DATA_BLOCK "LBP_Axis30"   // DB60
TITLE = Axis-specific signals / Signaux spécifiques à un axe
{ S7_Optimized_Access := 'FALSE' }
AUTHOR : SINUMERIK
FAMILY : SINUMERIK_ONE
VERSION : 6.24
// Interface between user program and axis/spindle, contains signals from/to axis/spindle 30 / Interface entre programme utilisateur et axe/broche, contient des signaux de/vers axe/broche 30
// stored: AutoNumber false, InstanceOfName LBP_typeAxisX, InstanceOfType UDT
"LBP_typeAxisX"
BEGIN
END_DATA_BLOCK

DATA_BLOCK "LBP_Axis31"   // DB61
TITLE = Axis-specific signals / Signaux spécifiques à un axe
{ S7_Optimized_Access := 'FALSE' }
AUTHOR : SINUMERIK
FAMILY : SINUMERIK_ONE
VERSION : 6.24
// Interface between user program and axis/spindle, contains signals from/to axis/spindle 31 / Interface entre programme utilisateur et axe/broche, contient des signaux de/vers axe/broche 31
// stored: AutoNumber false, InstanceOfName LBP_typeAxisX, InstanceOfType UDT
"LBP_typeAxisX"
BEGIN
END_DATA_BLOCK

DATA_BLOCK "LBP_Chan1"   // DB21
TITLE = Channel-specific signals / Signaux spécifiques à un canal
{ S7_Optimized_Access := 'FALSE' }
AUTHOR : SINUMERIK
FAMILY : SINUMERIK_ONE
VERSION : 6.24
// Interface between user program and channel, contains signals from/to channel 1 / Interface entre programme utilisateur et canal, contient des signaux de/vers canal 1
// stored: AutoNumber false, InstanceOfName LBP_typeChanX, InstanceOfType UDT
"LBP_typeChanX"
BEGIN
END_DATA_BLOCK

DATA_BLOCK "LBP_Chan10"   // DB30
TITLE = Channel-specific signals / Signaux spécifiques à un canal
{ S7_Optimized_Access := 'FALSE' }
AUTHOR : SINUMERIK
FAMILY : SINUMERIK_ONE
VERSION : 6.24
// Interface between user program and channel, contains signals from/to channel 10 / Interface entre programme utilisateur et canal, contient des signaux de/vers canal 10
// stored: AutoNumber false, InstanceOfName LBP_typeChanX, InstanceOfType UDT
"LBP_typeChanX"
BEGIN
END_DATA_BLOCK

DATA_BLOCK "LBP_Chan2"   // DB22
TITLE = Channel-specific signals / Signaux spécifiques à un canal
{ S7_Optimized_Access := 'FALSE' }
AUTHOR : SINUMERIK
FAMILY : SINUMERIK_ONE
VERSION : 6.24
// Interface between user program and channel, contains signals from/to channel 2 / Interface entre programme utilisateur et canal, contient des signaux de/vers canal 2
// stored: AutoNumber false, InstanceOfName LBP_typeChanX, InstanceOfType UDT
"LBP_typeChanX"
BEGIN
END_DATA_BLOCK

DATA_BLOCK "LBP_Chan3"   // DB23
TITLE = Channel-specific signals / Signaux spécifiques à un canal
{ S7_Optimized_Access := 'FALSE' }
AUTHOR : SINUMERIK
FAMILY : SINUMERIK_ONE
VERSION : 6.24
// Interface between user program and channel, contains signals from/to channel 3 / Interface entre programme utilisateur et canal, contient des signaux de/vers canal 3
// stored: AutoNumber false, InstanceOfName LBP_typeChanX, InstanceOfType UDT
"LBP_typeChanX"
BEGIN
END_DATA_BLOCK

DATA_BLOCK "LBP_Chan4"   // DB24
TITLE = Channel-specific signals / Signaux spécifiques à un canal
{ S7_Optimized_Access := 'FALSE' }
AUTHOR : SINUMERIK
FAMILY : SINUMERIK_ONE
VERSION : 6.24
// Interface between user program and channel, contains signals from/to channel 4 / Interface entre programme utilisateur et canal, contient des signaux de/vers canal 4
// stored: AutoNumber false, InstanceOfName LBP_typeChanX, InstanceOfType UDT
"LBP_typeChanX"
BEGIN
END_DATA_BLOCK

DATA_BLOCK "LBP_Chan5"   // DB25
TITLE = Channel-specific signals / Signaux spécifiques à un canal
{ S7_Optimized_Access := 'FALSE' }
AUTHOR : SINUMERIK
FAMILY : SINUMERIK_ONE
VERSION : 6.24
// Interface between user program and channel, contains signals from/to channel 5 / Interface entre programme utilisateur et canal, contient des signaux de/vers canal 5
// stored: AutoNumber false, InstanceOfName LBP_typeChanX, InstanceOfType UDT
"LBP_typeChanX"
BEGIN
END_DATA_BLOCK

DATA_BLOCK "LBP_Chan6"   // DB26
TITLE = Channel-specific signals / Signaux spécifiques à un canal
{ S7_Optimized_Access := 'FALSE' }
AUTHOR : SINUMERIK
FAMILY : SINUMERIK_ONE
VERSION : 6.24
// Interface between user program and channel, contains signals from/to channel 6 / Interface entre programme utilisateur et canal, contient des signaux de/vers canal 6
// stored: AutoNumber false, InstanceOfName LBP_typeChanX, InstanceOfType UDT
"LBP_typeChanX"
BEGIN
END_DATA_BLOCK

DATA_BLOCK "LBP_Chan7"   // DB27
TITLE = Channel-specific signals / Signaux spécifiques à un canal
{ S7_Optimized_Access := 'FALSE' }
AUTHOR : SINUMERIK
FAMILY : SINUMERIK_ONE
VERSION : 6.24
// Interface between user program and channel, contains signals from/to channel 7 / Interface entre programme utilisateur et canal, contient des signaux de/vers canal 7
// stored: AutoNumber false, InstanceOfName LBP_typeChanX, InstanceOfType UDT
"LBP_typeChanX"
BEGIN
END_DATA_BLOCK

DATA_BLOCK "LBP_Chan8"   // DB28
TITLE = Channel-specific signals / Signaux spécifiques à un canal
{ S7_Optimized_Access := 'FALSE' }
AUTHOR : SINUMERIK
FAMILY : SINUMERIK_ONE
VERSION : 6.24
// Interface between user program and channel, contains signals from/to channel 8 / Interface entre programme utilisateur et canal, contient des signaux de/vers canal 8
// stored: AutoNumber false, InstanceOfName LBP_typeChanX, InstanceOfType UDT
"LBP_typeChanX"
BEGIN
END_DATA_BLOCK

DATA_BLOCK "LBP_Chan9"   // DB29
TITLE = Channel-specific signals / Signaux spécifiques à un canal
{ S7_Optimized_Access := 'FALSE' }
AUTHOR : SINUMERIK
FAMILY : SINUMERIK_ONE
VERSION : 6.24
// Interface between user program and channel, contains signals from/to channel 9 / Interface entre programme utilisateur et canal, contient des signaux de/vers canal 9
// stored: AutoNumber false, InstanceOfName LBP_typeChanX, InstanceOfType UDT
"LBP_typeChanX"
BEGIN
END_DATA_BLOCK

DATA_BLOCK "LBP_ConfigData"   // DB7
TITLE = Configuration parameter
{ S7_Optimized_Access := 'FALSE' }
AUTHOR : SINUMERIK
FAMILY : SINUMERIK_ONE
VERSION : 6.14
// Contains parameters for the configuration and initialization of the basic program
// stored: AutoNumber false, InstanceOfName LBP_typeConfigData, InstanceOfType UDT
"LBP_typeConfigData"
BEGIN
END_DATA_BLOCK

DATA_BLOCK "LBP_HMI"   // DB19
TITLE = Operator panel signals / Signaux pupitre opérateur
{ S7_Optimized_Access := 'FALSE' }
AUTHOR : SINUMERIK
FAMILY : SINUMERIK_ONE
VERSION : 6.24
// Interface between user program and operator panel, contains signals from/to the operating software. / Interface entre programme utilisateur et pupitre opérateur, contient des signaux de/vers le logiciel d'exploitation.
// stored: AutoNumber false, InstanceOfName LBP_typeHMI, InstanceOfType UDT
"LBP_typeHMI"
BEGIN
END_DATA_BLOCK

DATA_BLOCK "LBP_ModeGroup"   // DB11
TITLE = Mode group signals / Signaux groupe de modes de fonctionnement
{ S7_Optimized_Access := 'FALSE' }
AUTHOR : SINUMERIK
FAMILY : SINUMERIK_ONE
VERSION : 6.24
// Interface between user program and mode groups, contains signals from/to the NC and operating software / Interface entre programme utilisateur et les groupes de modes de fonctionnement, contient des signaux de/vers le logiciel d'exploitation
// stored: AutoNumber false, InstanceOfName LBP_typeModeGroup, InstanceOfType UDT
"LBP_typeModeGroup"
BEGIN
END_DATA_BLOCK

DATA_BLOCK "LBP_NC"   // DB10
TITLE = NC signals / Signaux CN
{ S7_Optimized_Access := 'FALSE' }
AUTHOR : SINUMERIK
FAMILY : SINUMERIK_ONE
VERSION : 6.24
// Interface between user program and NC, contains signals from/to the NC, PLC and operating software. / Interface entre programme utilisateur et CN, contient des signaux de/vers CN, AP et logiciel d'exploitation.
// stored: AutoNumber false, InstanceOfName LBP_typeNC, InstanceOfType UDT
"LBP_typeNC"
BEGIN
END_DATA_BLOCK

DATA_BLOCK "LBP_OpUnitComm_DB"   // DB70
// stored: InstanceOfName LBP_OpUnitComm, InstanceOfType FB
"LBP_OpUnitComm"
   // VAR_OUTPUT
   //    Error : Bool;
   //    Status : Word;
   // END_VAR
   // VAR_IN_OUT
   //    Config : Variant;
   // END_VAR
   // VAR
   //    s_OpUnitConnInstance { S7_SetPoint := 'True'} : Array[1..6] of "LBP_InternalProc2";
   //    s_OpUnitNumber : UInt;
   //    s_OpUnitHardwareInterfaceId : HW_ANY;
   //    s_OpUnitEnabled : Array[1..6] of Bool;
   //    s_OpUnitConfig { S7_SetPoint := 'True'} : Array[1..6] of "LBP_typeInternal1";
   //    s_OpUnitControlMcp : Array[1..5] of Struct
   //       active : Bool;
   //       stop : Bool;
   //       notSend : Bool;
   //       connected : Bool;
   //       warning : Bool;
   //       error : Bool;
   //       status : Word;
   //       info : Word;
   //       alert : Bool;
   //       alertDelay { S7_SetPoint := 'True'} : TON_TIME;
   //    END_STRUCT;
   //    s_OpUnitControlIdent : Struct
   //       strobe : Bool;
   //       busAddress : USInt;
   //       modeDck : Bool;
   //       numberOfInputBytes : UInt;
   //       numberOfOutputBytes : UInt;
   //       mcpType : Word;
   //       done : Bool;
   //       error : Bool;
   //       status : Word;
   //       info : Word;
   //    END_STRUCT;
   //    s_OpUnitData : Array[1..6] of Struct
   //       connect : Bool;
   //       ident : Bool;
   //       notSend : Bool;
   //       busy : Bool;
   //       connected : Bool;
   //       warning : Bool;
   //       error : Bool;
   //       identReady : Bool;
   //       reconnect : Bool;
   //       status : Word;
   //       errorInfo : Word;
   //       mcpType : Word;
   //       mcpDipFixes : Word;
   //       numberOfOutputBytes : UInt;
   //       numberOfInputBytes : UInt;
   //       numberOfHandwheels : UInt;
   //       handwheelRecent : Bool;
   //       handwheelPulses1 : Int;
   //       handwheelPulses2 : Int;
   //       handwheelStopped1 : Bool;
   //       handwheelStopped2 : Bool;
   //       reconnectTimer { S7_SetPoint := 'True'} : TON_TIME;
   //       reconnectCounter : UInt;
   //    END_STRUCT;
   //    s_init : Bool;
   //    statReadWriteRecordActive : Bool;
   //    statReadWriteRecordComplete : Bool;
   //    statReadWriteRecordAbort : Bool;
   //    statReadWriteRecordMcp : UInt;
   //    statReadWriteRecordTimeout : TON_TIME;
   //    statReadWriteRecordData { S7_SetPoint := 'True'} : "LBP_typeInternal5";
   // END_VAR
BEGIN
END_DATA_BLOCK

DATA_BLOCK "LBP_TMLoad"   // DB71
TITLE = Tool management / Gestion des outils
{ S7_Optimized_Access := 'FALSE' }
AUTHOR : SINUMERIK
FAMILY : SINUMERIK_ONE
VERSION : 6.24
// Interface between user program and tool management, contains signals from/to Load/Unload magazine / Interface entre programme utilisateur et gestion d'outil, contient des signaux de/vers Chargement/déchargement de magasin
// stored: AutoNumber false, InstanceOfName LBP_typeTMLoad, InstanceOfType UDT
"LBP_typeTMLoad"
BEGIN
END_DATA_BLOCK

DATA_BLOCK "LBP_TMLoadMT"   // DB1071
TITLE = Tool management / Gestion des outils
{ S7_Optimized_Access := 'FALSE' }
AUTHOR : SINUMERIK
FAMILY : SINUMERIK_ONE
VERSION : 6.24
// Interface between user program and tool management, contains signals from/to Load/Unload magazine (multitool). / Interface entre programme utilisateur et gestion d'outil, contient des signaux de/vers Chargement/déchargement de magasin (Multitool).
// stored: AutoNumber false, InstanceOfName LBP_typeTMLoadMT, InstanceOfType UDT
"LBP_typeTMLoadMT"
BEGIN
END_DATA_BLOCK

DATA_BLOCK "LBP_TMSpindle"   // DB72
TITLE = Tool management / Gestion des outils
{ S7_Optimized_Access := 'FALSE' }
AUTHOR : SINUMERIK
FAMILY : SINUMERIK_ONE
VERSION : 6.24
// Interface between user program and tool management, contains signals for spindle as change position. / Interface entre programme utilisateur et gestion d'outil, contient des signaux pour broche en tant que position de changement.
// stored: AutoNumber false, InstanceOfName LBP_typeTMSpindle, InstanceOfType UDT
"LBP_typeTMSpindle"
BEGIN
END_DATA_BLOCK

DATA_BLOCK "LBP_TMSpindleMT"   // DB1072
TITLE = Tool management / Gestion des outils
{ S7_Optimized_Access := 'FALSE' }
AUTHOR : SINUMERIK
FAMILY : SINUMERIK_ONE
VERSION : 6.24
// Interface between user program and tool management, contains signals for spindle as change position (multitool). / Interface entre programme utilisateur et gestion d'outil, contient des signaux pour broche en tant que position de changement (Multitool).
// stored: AutoNumber false, InstanceOfName LBP_typeTMSpindleMT, InstanceOfType UDT
"LBP_typeTMSpindleMT"
BEGIN
END_DATA_BLOCK

DATA_BLOCK "LBP_TMTurret"   // DB73
TITLE = Tool management / Gestion des outils
{ S7_Optimized_Access := 'FALSE' }
AUTHOR : SINUMERIK
FAMILY : SINUMERIK_ONE
VERSION : 6.24
// Interface between user program and tool management, contains signals for turret. / Interface entre programme utilisateur et gestion d'outil, contient des signaux pour tourelle.
// stored: AutoNumber false, InstanceOfName LBP_typeTMTurret, InstanceOfType UDT
"LBP_typeTMTurret"
BEGIN
END_DATA_BLOCK

DATA_BLOCK "LBP_TMTurretMT"   // DB1073
TITLE = Tool management / Gestion des outils
{ S7_Optimized_Access := 'FALSE' }
AUTHOR : SINUMERIK
FAMILY : SINUMERIK_ONE
VERSION : 6.24
// Interface between user program and tool management, contains signals for turret (multitool). / Interface entre programme utilisateur et gestion d'outil, contient des signaux pour tourelle (Multitool).
// stored: AutoNumber false, InstanceOfName LBP_typeTMTurretMT, InstanceOfType UDT
"LBP_typeTMTurretMT"
BEGIN
END_DATA_BLOCK

DATA_BLOCK "LBP_Internal2"   // DB25001
TITLE = Internal DB for basic program / DB interne pour programme de base
// DB only for internal use in the basic program / DB réservé à l'utilisation interne dans le programme de base
// stored: InstanceOfName LBP_InternalProc7, InstanceOfType FB
"LBP_InternalProc7"
   // VAR_OUTPUT
   //    error { ExternalAccessible := 'False'; ExternalVisible := 'False'; ExternalWritable := 'False'} : Bool;
   // END_VAR
   // VAR
   //    statTimer1 { ExternalAccessible := 'False'; ExternalVisible := 'False'; ExternalWritable := 'False'} : Array[1..8] of IEC_TIMER;
   //    statTimer2 { ExternalAccessible := 'False'; ExternalVisible := 'False'; ExternalWritable := 'False'} : Array[1..8] of IEC_TIMER;
   //    statTimerActivationImmediately { ExternalAccessible := 'False'; ExternalVisible := 'False'; ExternalWritable := 'False'} : Array[1..8] of IEC_TIMER;   // Delay time for immediate activation / Temporisation pour activation immédiate
   //    statActivationImmediately { ExternalAccessible := 'False'; ExternalVisible := 'False'; ExternalWritable := 'False'} : Array[1..8] of Bool;
   //    statImpReloadT2 { ExternalAccessible := 'False'; ExternalVisible := 'False'; ExternalWritable := 'False'} : Array[1..8] of R_TRIG;
   //    statMcp1 { ExternalAccessible := 'False'; ExternalVisible := 'False'; ExternalWritable := 'False'} : Array[0..1, 0..7] of Byte;   // Image of mcp1 to detect any changes / Image de la mcp1 pour comparaison
   //    statMcp2 { ExternalAccessible := 'False'; ExternalVisible := 'False'; ExternalWritable := 'False'} : Array[0..1, 0..7] of Byte;   // Image of mcp2 to detect any changes / Image de la mcp2 pour comparaison
   //    statTimerDataTranfer { ExternalAccessible := 'False'; ExternalVisible := 'False'; ExternalWritable := 'False'} : IEC_TIMER;
   //    statChanInReset { ExternalAccessible := 'False'; ExternalVisible := 'False'; ExternalWritable := 'False'} : Array[1..10] of Bool;
   //    statAktProfile { ExternalAccessible := 'False'; ExternalVisible := 'False'; ExternalWritable := 'False'} : Struct
   //       ESaveOn : Bool;   // Activate energy-saving profile immediately / Activer immédiatement le profil d'économie d'énergie
   //       ReloadT2 : Bool;   // Reload Prewarning time (T2) / Recharger temps de préavis (T2)
   //       res0_2 : Bool;
   //       res0_3 : Bool;
   //       res0_4 : Bool;
   //       res0_5 : Bool;
   //       res0_6 : Bool;
   //       res0_7 : Bool;
   //       HmiESaveOn : Bool;   // HMI->PLC: Activate energy-saving profile immediately / IHM->AP : activer immédiatement le profil d'économie d'énergie
   //       res1_1 : Bool;
   //       res1_2 : Bool;
   //       res1_3 : Bool;
   //       res1_4 : Bool;
   //       res1_5 : Bool;
   //       res1_6 : Bool;
   //       res1_7 : Bool;
   //       MasterCompSig : Bool;   // Master computer signal / Signal ordinateur maître
   //       PlcUserSig : Bool;   // PLC user signal / AP signal utilisateur
   //       res2_2 : Bool;
   //       res2_3 : Bool;
   //       res2_4 : Bool;
   //       res2_5 : Bool;
   //       res2_6 : Bool;
   //       res2_7 : Bool;
   //       res3 : Byte;
   //       ESaveIsOn : Bool;   // Energy-saving state active / État économie d'énergie actif
   //       T1Expired : Bool;   // Activation time T1 expired / Temps d'activation T1 écoulé
   //       res4_2 : Bool;
   //       res4_3 : Bool;
   //       res4_4 : Bool;
   //       res4_5 : Bool;
   //       res4_6 : Bool;
   //       res4_7 : Bool;
   //       res5 : Byte;
   //       ActValT1 : Int;   // T1 current value / T1 valeur réelle
   //       ActValT2 : Int;   // T2 current value / T2 valeur réelle
   //       ESaveValid : Bool;   // HMI->PLC: Energy-saving profile valid / IHM->AP : profil d'économie d'énergie valide
   //       ESaveOff : Bool;   // HMI->PLC: Deactivate energy-saving profileblock energy-saving profile / IHM->AP : désactiver/bloquer le profil d'économie d'énergie
   //       res10_2 : Bool;
   //       res10_3 : Bool;
   //       res10_4 : Bool;
   //       res10_5 : Bool;
   //       res10_6 : Bool;
   //       res10_7 : Bool;
   //       CondOpPanel : Bool;   // HMI->PLC: Operator panel / IHM->AP : pupitre opérateur
   //       CondDataTransfer : Bool;   // HMI->PLC: Data transfer / IHM->AP : transmission de données
   //       CondWindowChange : Bool;   // HMI->PLC: Window change / IHM->AP : changement de fenêtre
   //       res11_3 : Bool;
   //       res11_4 : Bool;
   //       res11_5 : Bool;
   //       res11_6 : Bool;
   //       res11_7 : Bool;
   //       CondMCP : Bool;   // HMI->PLC: Machine control panel / IHM->AP : pupitre opérateur machine
   //       res12_1 : Bool;
   //       res12_2 : Bool;
   //       res12_3 : Bool;
   //       res12_4 : Bool;
   //       res12_5 : Bool;
   //       res12_6 : Bool;
   //       res12_7 : Bool;
   //       CondNcChan1 : Bool;   // HMI->PLC: NC channel 1 in reset / IHM->AP : canal CN 1 en Reset
   //       CondNcChan2 : Bool;   // HMI->PLC: NC channel 2 in reset / IHM->AP : canal CN 2 en Reset
   //       CondNcChan3 : Bool;   // HMI->PLC: NC channel 3 in reset / IHM->AP : canal CN 3 en Reset
   //       CondNcChan4 : Bool;   // HMI->PLC: NC channel 4 in reset / IHM->AP : canal CN 4 en Reset
   //       CondNcChan5 : Bool;   // HMI->PLC: NC channel 5 in reset / IHM->AP : canal CN 5 en Reset
   //       CondNcChan6 : Bool;   // HMI->PLC: NC channel 6 in reset / IHM->AP : canal CN 6 en Reset
   //       CondNcChan7 : Bool;   // HMI->PLC: NC channel 7 in reset / IHM->AP : canal CN 7 en Reset
   //       CondNcChan8 : Bool;   // HMI->PLC: NC channel 8 in reset / IHM->AP : canal CN 8 en Reset
   //       CondNcChan9 : Bool;   // HMI->PLC: NC channel 9 in reset / IHM->AP : canal CN 9 en Reset
   //       CondNcChan10 : Bool;   // HMI->PLC: NC channel 10 in reset / IHM->AP : canal CN 10 en Reset
   //       res14_2 : Bool;
   //       res14_3 : Bool;
   //       res14_4 : Bool;
   //       res14_5 : Bool;
   //       res14_6 : Bool;
   //       res14_7 : Bool;
   //       CondMasterCompSig : Bool;   // HMI->PLC: Master computer signal / IHM->AP : signal ordinateur maître
   //       CondPlcUserSig : Bool;   // HMI->PLC: PLC user signal / IHM->AP : signal utilisateur AP
   //       res15_2 : Bool;
   //       res15_3 : Bool;
   //       res15_4 : Bool;
   //       res15_5 : Bool;
   //       res15_6 : Bool;
   //       res15_7 : Bool;
   //       PresetT1 : Int;   // HMI->PLC: Activation time T1 / IHM->AP : temps d'activation T1
   //       PresetT2 : Int;   // HMI->PLC: Activation time T2 / IHM->AP : temps d'activation T2
   //    END_STRUCT;
   // END_VAR
BEGIN
END_DATA_BLOCK

DATA_BLOCK "LBP_Internal3"   // DB25002
TITLE = Internal DB for basic program / DB interne pour programme de base
// DB only for internal use in the basic program / DB réservé à l'utilisation interne dans le programme de base
// stored: InstanceOfName LBP_InternalProc8, InstanceOfType FB
"LBP_InternalProc8"
   // VAR
   //    statPlcCtrlsNm1 { ExternalAccessible := 'False'; ExternalVisible := 'False'; ExternalWritable := 'False'} : Bool;
   //    statDateAndTime { ExternalAccessible := 'False'; ExternalVisible := 'False'; ExternalWritable := 'False'} : Date_And_Time;
   //    statLastSecond { ExternalAccessible := 'False'; ExternalVisible := 'False'; ExternalWritable := 'False'} : Byte;
   // END_VAR
BEGIN
END_DATA_BLOCK

DATA_BLOCK "LBP_Internal9"   // DB25005
TITLE = Internal DB for basic program / DB interne pour programme de base
// DB only for internal use in the basic program / DB réservé à l'utilisation interne dans le programme de base
// stored: InstanceOfName LBP_InternalProc9, InstanceOfType FB
"LBP_InternalProc9"
   // VAR
   //    statSymbols { ExternalAccessible := 'False'; ExternalVisible := 'False'; ExternalWritable := 'False'} : Array[0..31] of WString;
   //    statResolvedSymbols { ExternalAccessible := 'False'; ExternalVisible := 'False'; ExternalWritable := 'False'} : Array[0..31] of ResolvedSymbol;
   //    InstResolveSymbols { ExternalAccessible := 'False'; ExternalVisible := 'False'; ExternalWritable := 'False'} : ResolveSymbols;
   //    statDestOffsets { ExternalAccessible := 'False'; ExternalVisible := 'False'; ExternalWritable := 'False'} : Array[0..31] of DInt;
   //    statResolveExecute { ExternalAccessible := 'False'; ExternalVisible := 'False'; ExternalWritable := 'False'} : Bool;
   //    statResolveProcessing { ExternalAccessible := 'False'; ExternalVisible := 'False'; ExternalWritable := 'False'} : Bool;
   //    statResolveError { ExternalAccessible := 'False'; ExternalVisible := 'False'; ExternalWritable := 'False'} : Bool;
   //    statResolveStatus { ExternalAccessible := 'False'; ExternalVisible := 'False'; ExternalWritable := 'False'} : Word;
   //    statReResolveNeeded { ExternalAccessible := 'False'; ExternalVisible := 'False'; ExternalWritable := 'False'} : Array[0..31] of Bool;
   // END_VAR
BEGIN
END_DATA_BLOCK

DATA_BLOCK "LBP_InternalDB1020"   // DB1020
TITLE = Internal DB for basic program / DB interne pour programme de base
// DB only for internal use in the basic program / DB réservé à l'utilisation interne dans le programme de base
// stored: AutoNumber false, InstanceOfName LBP_InternalFB1020, InstanceOfType FB
"LBP_InternalFB1020"
   // VAR_INPUT
   //    IN1 : UDInt;
   //    IN2 : UDInt;
   //    IN3 : Word;
   //    IN4 : Variant;
   //    IN5 : Variant;
   //    IN6 : Variant;
   //    IN7 : Variant;
   //    IN8 : Variant;
   //    IN9 : Variant;
   //    IN10 : Variant;
   //    IN11 : Variant;
   //    IN12 : Variant;
   // END_VAR
   // VAR_OUTPUT
   //    OUT1 : Bool;
   //    OUT2 : DWord;
   //    OUT3 : UInt;
   // END_VAR
   // VAR
   //    LBP_AlarmType_ErrMsg { S7_SetPoint := 'True'} : Diag_Alarm;
   //    LBP_AlarmType_OpMsg { S7_SetPoint := 'True'} : Diag_Alarm;
   //    LBP_AlarmType_InfoMsg { S7_SetPoint := 'True'} : Diag_Alarm;
   //    LBP_DB2AlarmType_ErrMsg { S7_SetPoint := 'True'} : Diag_Alarm;
   //    LBP_DB2AlarmType_OpMsg { S7_SetPoint := 'True'} : Diag_Alarm;
   //    LBP_DB2AlarmType_InfoMsg { S7_SetPoint := 'True'} : Diag_Alarm;
   //    LBP_UserAlarmType_ErrMsg { S7_SetPoint := 'True'} : Diag_Alarm;
   //    LBP_UserAlarmType_OpMsg { S7_SetPoint := 'True'} : Diag_Alarm;
   //    LBP_UserAlarmType_InfoMsg { S7_SetPoint := 'True'} : Diag_Alarm;
   //    LBP_UserAlarmType_AckMsg { S7_SetPoint := 'True'} : Diag_Alarm;
   //    s_strct_DB2AddressLastCycle : Struct
   //       LwByteAddress : DInt;
   //       LwBitAddress : DInt;
   //    END_STRUCT;
   //    s_DB2_MaxScanByteUser : DInt;
   //    s_DB7_Params : Struct
   //       MaxAxis : Int;
   //       MaxChan : Int;
   //       MsgUser : Int;
   //       ExtendChanAxMsg : Bool;
   //       ActivChan : Array[1..10] of Bool;
   //       ActivAxis : Array[1..31] of Bool;
   //    END_STRUCT;
   //    s_firstScanFinished : Bool;
   //    s_FC10_Quit : Struct
   //       QuitEdge : Bool;
   //       LwByteAddress : DInt;
   //       DB2ScanFinished : Bool;
   //    END_STRUCT;
   //    s_CounterActiveDB2Alarms : UInt;
   //    s_FC10_ToUserIf_OLD : Bool;
   // END_VAR
BEGIN
END_DATA_BLOCK

DATA_BLOCK "LBP_InternalDB3"   // DB3
TITLE = PLC-Error / Messages / Erreur AP / messages
{ S7_Optimized_Access := 'FALSE' }
AUTHOR : SINUMERIK
FAMILY : SINUMERIK_ONE
VERSION : 6.24
// DB only for internal use in the basic program / DB réservé à l'utilisation interne dans le programme de base
// stored: AutoNumber false, InstanceOfName LBP_typeAlarmMsgs, InstanceOfType UDT
"LBP_typeAlarmMsgs"
BEGIN
END_DATA_BLOCK

DATA_BLOCK "DB_AnalogInputs"   // DB2200
// stored: AutoNumber false, InstanceOfName FB_AnalogInputs, InstanceOfType FB
"FB_AnalogInputs"
BEGIN
END_DATA_BLOCK

DATA_BLOCK "DB_DigitalInputs"   // DB2210
// stored: AutoNumber false, InstanceOfName FB_DigitalInputs, InstanceOfType FB
"FB_DigitalInputs"
BEGIN
END_DATA_BLOCK

DATA_BLOCK "DB_DigitalInputsBW_Station"   // DB2214
// stored: AutoNumber false, InstanceOfName FB_DigitalInputsBW_Station, InstanceOfType FB
"FB_DigitalInputsBW_Station"
BEGIN
END_DATA_BLOCK

DATA_BLOCK "DB_DigitalInputsSonplas"   // DB2211
// stored: AutoNumber false, InstanceOfName FB_DigitalInputsSonplas, InstanceOfType FB
"FB_DigitalInputsSonplas"
BEGIN
END_DATA_BLOCK

DATA_BLOCK "DB_AnalogOutputs"   // DB2113
// stored: AutoNumber false, InstanceOfName FB_AnalogOutputs, InstanceOfType FB
"FB_AnalogOutputs"
BEGIN
END_DATA_BLOCK

DATA_BLOCK "DB_DigitalOutputs"   // DB2103
// stored: AutoNumber false, InstanceOfName FB_DigitalOutputs, InstanceOfType FB
"FB_DigitalOutputs"
BEGIN
END_DATA_BLOCK

DATA_BLOCK "DB_DigitalOutputsSonplas"   // DB2104
// stored: AutoNumber false, InstanceOfName FB_DigitalOutputsSonplas, InstanceOfType FB
"FB_DigitalOutputsSonplas"
BEGIN
END_DATA_BLOCK

DATA_BLOCK "F-DB_DigitalInputs"   // DB110, F_DB
// stored: AutoNumber false, InstanceOfName F-FB_DigitalInput, InstanceOfType FB
"F-FB_DigitalInput"
BEGIN
END_DATA_BLOCK

DATA_BLOCK "F-DB_DigitalOutput"   // DB111, F_DB
// stored: AutoNumber false, InstanceOfName F-FB_DigitalOutput, InstanceOfType FB
"F-FB_DigitalOutput"
BEGIN
END_DATA_BLOCK

DATA_BLOCK "LBP_ReadVar_DB_Axis01_X"   // DB4101
// stored: AutoNumber false, InstanceOfName LBP_ReadVar, InstanceOfType FB
"LBP_ReadVar"
   // VAR_INPUT
   //    Req : Bool;
   //    NumVar : Int;
   //    Addr1 : Variant;
   //    Unit1 : Byte;
   //    Column1 : Word;
   //    Line1 : Word;
   //    Addr2 : Variant;
   //    Unit2 : Byte;
   //    Column2 : Word;
   //    Line2 : Word;
   //    Addr3 : Variant;
   //    Unit3 : Byte;
   //    Column3 : Word;
   //    Line3 : Word;
   //    Addr4 : Variant;
   //    Unit4 : Byte;
   //    Column4 : Word;
   //    Line4 : Word;
   //    Addr5 : Variant;
   //    Unit5 : Byte;
   //    Column5 : Word;
   //    Line5 : Word;
   //    Addr6 : Variant;
   //    Unit6 : Byte;
   //    Column6 : Word;
   //    Line6 : Word;
   //    Addr7 : Variant;
   //    Unit7 : Byte;
   //    Column7 : Word;
   //    Line7 : Word;
   //    Addr8 : Variant;
   //    Unit8 : Byte;
   //    Column8 : Word;
   //    Line8 : Word;
   // END_VAR
   // VAR_OUTPUT
   //    Error : Bool;
   //    NDR : Bool;
   //    State : Word;
   // END_VAR
   // VAR_IN_OUT
   //    RD1 : Variant;
   //    RD2 : Variant;
   //    RD3 : Variant;
   //    RD4 : Variant;
   //    RD5 : Variant;
   //    RD6 : Variant;
   //    RD7 : Variant;
   //    RD8 : Variant;
   // END_VAR
   // VAR
   //    ident : Byte;
   //    regist : Bool;
   //    flanke : Bool;
   //    progtest : Bool;
   //    err_cls_cod : Word;
   //    err_stat : Word;
   //    s_fifoRef : UInt;
   //    s_Reserved1 : Word;
   //    s_Reserved2 : DWord;
   //    s_Reserved3 : DWord;
   // END_VAR
BEGIN
END_DATA_BLOCK

DATA_BLOCK "LBP_ReadVar_DB_Axis02_Y"   // DB4102
// stored: AutoNumber false, InstanceOfName LBP_ReadVar, InstanceOfType FB
"LBP_ReadVar"
   // VAR_INPUT
   //    Req : Bool;
   //    NumVar : Int;
   //    Addr1 : Variant;
   //    Unit1 : Byte;
   //    Column1 : Word;
   //    Line1 : Word;
   //    Addr2 : Variant;
   //    Unit2 : Byte;
   //    Column2 : Word;
   //    Line2 : Word;
   //    Addr3 : Variant;
   //    Unit3 : Byte;
   //    Column3 : Word;
   //    Line3 : Word;
   //    Addr4 : Variant;
   //    Unit4 : Byte;
   //    Column4 : Word;
   //    Line4 : Word;
   //    Addr5 : Variant;
   //    Unit5 : Byte;
   //    Column5 : Word;
   //    Line5 : Word;
   //    Addr6 : Variant;
   //    Unit6 : Byte;
   //    Column6 : Word;
   //    Line6 : Word;
   //    Addr7 : Variant;
   //    Unit7 : Byte;
   //    Column7 : Word;
   //    Line7 : Word;
   //    Addr8 : Variant;
   //    Unit8 : Byte;
   //    Column8 : Word;
   //    Line8 : Word;
   // END_VAR
   // VAR_OUTPUT
   //    Error : Bool;
   //    NDR : Bool;
   //    State : Word;
   // END_VAR
   // VAR_IN_OUT
   //    RD1 : Variant;
   //    RD2 : Variant;
   //    RD3 : Variant;
   //    RD4 : Variant;
   //    RD5 : Variant;
   //    RD6 : Variant;
   //    RD7 : Variant;
   //    RD8 : Variant;
   // END_VAR
   // VAR
   //    ident : Byte;
   //    regist : Bool;
   //    flanke : Bool;
   //    progtest : Bool;
   //    err_cls_cod : Word;
   //    err_stat : Word;
   //    s_fifoRef : UInt;
   //    s_Reserved1 : Word;
   //    s_Reserved2 : DWord;
   //    s_Reserved3 : DWord;
   // END_VAR
BEGIN
END_DATA_BLOCK

DATA_BLOCK "LBP_ReadVar_DB_Axis03_ZM"   // DB4103
// stored: AutoNumber false, InstanceOfName LBP_ReadVar, InstanceOfType FB
"LBP_ReadVar"
   // VAR_INPUT
   //    Req : Bool;
   //    NumVar : Int;
   //    Addr1 : Variant;
   //    Unit1 : Byte;
   //    Column1 : Word;
   //    Line1 : Word;
   //    Addr2 : Variant;
   //    Unit2 : Byte;
   //    Column2 : Word;
   //    Line2 : Word;
   //    Addr3 : Variant;
   //    Unit3 : Byte;
   //    Column3 : Word;
   //    Line3 : Word;
   //    Addr4 : Variant;
   //    Unit4 : Byte;
   //    Column4 : Word;
   //    Line4 : Word;
   //    Addr5 : Variant;
   //    Unit5 : Byte;
   //    Column5 : Word;
   //    Line5 : Word;
   //    Addr6 : Variant;
   //    Unit6 : Byte;
   //    Column6 : Word;
   //    Line6 : Word;
   //    Addr7 : Variant;
   //    Unit7 : Byte;
   //    Column7 : Word;
   //    Line7 : Word;
   //    Addr8 : Variant;
   //    Unit8 : Byte;
   //    Column8 : Word;
   //    Line8 : Word;
   // END_VAR
   // VAR_OUTPUT
   //    Error : Bool;
   //    NDR : Bool;
   //    State : Word;
   // END_VAR
   // VAR_IN_OUT
   //    RD1 : Variant;
   //    RD2 : Variant;
   //    RD3 : Variant;
   //    RD4 : Variant;
   //    RD5 : Variant;
   //    RD6 : Variant;
   //    RD7 : Variant;
   //    RD8 : Variant;
   // END_VAR
   // VAR
   //    ident : Byte;
   //    regist : Bool;
   //    flanke : Bool;
   //    progtest : Bool;
   //    err_cls_cod : Word;
   //    err_stat : Word;
   //    s_fifoRef : UInt;
   //    s_Reserved1 : Word;
   //    s_Reserved2 : DWord;
   //    s_Reserved3 : DWord;
   // END_VAR
BEGIN
END_DATA_BLOCK

DATA_BLOCK "LBP_ReadVar_DB_Axis04_B"   // DB4109
// stored: AutoNumber false, InstanceOfName LBP_ReadVar, InstanceOfType FB
"LBP_ReadVar"
   // VAR_INPUT
   //    Req : Bool;
   //    NumVar : Int;
   //    Addr1 : Variant;
   //    Unit1 : Byte;
   //    Column1 : Word;
   //    Line1 : Word;
   //    Addr2 : Variant;
   //    Unit2 : Byte;
   //    Column2 : Word;
   //    Line2 : Word;
   //    Addr3 : Variant;
   //    Unit3 : Byte;
   //    Column3 : Word;
   //    Line3 : Word;
   //    Addr4 : Variant;
   //    Unit4 : Byte;
   //    Column4 : Word;
   //    Line4 : Word;
   //    Addr5 : Variant;
   //    Unit5 : Byte;
   //    Column5 : Word;
   //    Line5 : Word;
   //    Addr6 : Variant;
   //    Unit6 : Byte;
   //    Column6 : Word;
   //    Line6 : Word;
   //    Addr7 : Variant;
   //    Unit7 : Byte;
   //    Column7 : Word;
   //    Line7 : Word;
   //    Addr8 : Variant;
   //    Unit8 : Byte;
   //    Column8 : Word;
   //    Line8 : Word;
   // END_VAR
   // VAR_OUTPUT
   //    Error : Bool;
   //    NDR : Bool;
   //    State : Word;
   // END_VAR
   // VAR_IN_OUT
   //    RD1 : Variant;
   //    RD2 : Variant;
   //    RD3 : Variant;
   //    RD4 : Variant;
   //    RD5 : Variant;
   //    RD6 : Variant;
   //    RD7 : Variant;
   //    RD8 : Variant;
   // END_VAR
   // VAR
   //    ident : Byte;
   //    regist : Bool;
   //    flanke : Bool;
   //    progtest : Bool;
   //    err_cls_cod : Word;
   //    err_stat : Word;
   //    s_fifoRef : UInt;
   //    s_Reserved1 : Word;
   //    s_Reserved2 : DWord;
   //    s_Reserved3 : DWord;
   // END_VAR
BEGIN
END_DATA_BLOCK

DATA_BLOCK "LBP_ReadVar_DB_Axis05_U1"   // DB4104
// stored: AutoNumber false, InstanceOfName LBP_ReadVar, InstanceOfType FB
"LBP_ReadVar"
   // VAR_INPUT
   //    Req : Bool;
   //    NumVar : Int;
   //    Addr1 : Variant;
   //    Unit1 : Byte;
   //    Column1 : Word;
   //    Line1 : Word;
   //    Addr2 : Variant;
   //    Unit2 : Byte;
   //    Column2 : Word;
   //    Line2 : Word;
   //    Addr3 : Variant;
   //    Unit3 : Byte;
   //    Column3 : Word;
   //    Line3 : Word;
   //    Addr4 : Variant;
   //    Unit4 : Byte;
   //    Column4 : Word;
   //    Line4 : Word;
   //    Addr5 : Variant;
   //    Unit5 : Byte;
   //    Column5 : Word;
   //    Line5 : Word;
   //    Addr6 : Variant;
   //    Unit6 : Byte;
   //    Column6 : Word;
   //    Line6 : Word;
   //    Addr7 : Variant;
   //    Unit7 : Byte;
   //    Column7 : Word;
   //    Line7 : Word;
   //    Addr8 : Variant;
   //    Unit8 : Byte;
   //    Column8 : Word;
   //    Line8 : Word;
   // END_VAR
   // VAR_OUTPUT
   //    Error : Bool;
   //    NDR : Bool;
   //    State : Word;
   // END_VAR
   // VAR_IN_OUT
   //    RD1 : Variant;
   //    RD2 : Variant;
   //    RD3 : Variant;
   //    RD4 : Variant;
   //    RD5 : Variant;
   //    RD6 : Variant;
   //    RD7 : Variant;
   //    RD8 : Variant;
   // END_VAR
   // VAR
   //    ident : Byte;
   //    regist : Bool;
   //    flanke : Bool;
   //    progtest : Bool;
   //    err_cls_cod : Word;
   //    err_stat : Word;
   //    s_fifoRef : UInt;
   //    s_Reserved1 : Word;
   //    s_Reserved2 : DWord;
   //    s_Reserved3 : DWord;
   // END_VAR
BEGIN
END_DATA_BLOCK

DATA_BLOCK "LBP_ReadVar_DB_Axis06_U2"   // DB4106
// stored: AutoNumber false, InstanceOfName LBP_ReadVar, InstanceOfType FB
"LBP_ReadVar"
   // VAR_INPUT
   //    Req : Bool;
   //    NumVar : Int;
   //    Addr1 : Variant;
   //    Unit1 : Byte;
   //    Column1 : Word;
   //    Line1 : Word;
   //    Addr2 : Variant;
   //    Unit2 : Byte;
   //    Column2 : Word;
   //    Line2 : Word;
   //    Addr3 : Variant;
   //    Unit3 : Byte;
   //    Column3 : Word;
   //    Line3 : Word;
   //    Addr4 : Variant;
   //    Unit4 : Byte;
   //    Column4 : Word;
   //    Line4 : Word;
   //    Addr5 : Variant;
   //    Unit5 : Byte;
   //    Column5 : Word;
   //    Line5 : Word;
   //    Addr6 : Variant;
   //    Unit6 : Byte;
   //    Column6 : Word;
   //    Line6 : Word;
   //    Addr7 : Variant;
   //    Unit7 : Byte;
   //    Column7 : Word;
   //    Line7 : Word;
   //    Addr8 : Variant;
   //    Unit8 : Byte;
   //    Column8 : Word;
   //    Line8 : Word;
   // END_VAR
   // VAR_OUTPUT
   //    Error : Bool;
   //    NDR : Bool;
   //    State : Word;
   // END_VAR
   // VAR_IN_OUT
   //    RD1 : Variant;
   //    RD2 : Variant;
   //    RD3 : Variant;
   //    RD4 : Variant;
   //    RD5 : Variant;
   //    RD6 : Variant;
   //    RD7 : Variant;
   //    RD8 : Variant;
   // END_VAR
   // VAR
   //    ident : Byte;
   //    regist : Bool;
   //    flanke : Bool;
   //    progtest : Bool;
   //    err_cls_cod : Word;
   //    err_stat : Word;
   //    s_fifoRef : UInt;
   //    s_Reserved1 : Word;
   //    s_Reserved2 : DWord;
   //    s_Reserved3 : DWord;
   // END_VAR
BEGIN
END_DATA_BLOCK

DATA_BLOCK "LBP_ReadVar_DB_Axis07_V"   // DB4107
// stored: AutoNumber false, InstanceOfName LBP_ReadVar, InstanceOfType FB
"LBP_ReadVar"
   // VAR_INPUT
   //    Req : Bool;
   //    NumVar : Int;
   //    Addr1 : Variant;
   //    Unit1 : Byte;
   //    Column1 : Word;
   //    Line1 : Word;
   //    Addr2 : Variant;
   //    Unit2 : Byte;
   //    Column2 : Word;
   //    Line2 : Word;
   //    Addr3 : Variant;
   //    Unit3 : Byte;
   //    Column3 : Word;
   //    Line3 : Word;
   //    Addr4 : Variant;
   //    Unit4 : Byte;
   //    Column4 : Word;
   //    Line4 : Word;
   //    Addr5 : Variant;
   //    Unit5 : Byte;
   //    Column5 : Word;
   //    Line5 : Word;
   //    Addr6 : Variant;
   //    Unit6 : Byte;
   //    Column6 : Word;
   //    Line6 : Word;
   //    Addr7 : Variant;
   //    Unit7 : Byte;
   //    Column7 : Word;
   //    Line7 : Word;
   //    Addr8 : Variant;
   //    Unit8 : Byte;
   //    Column8 : Word;
   //    Line8 : Word;
   // END_VAR
   // VAR_OUTPUT
   //    Error : Bool;
   //    NDR : Bool;
   //    State : Word;
   // END_VAR
   // VAR_IN_OUT
   //    RD1 : Variant;
   //    RD2 : Variant;
   //    RD3 : Variant;
   //    RD4 : Variant;
   //    RD5 : Variant;
   //    RD6 : Variant;
   //    RD7 : Variant;
   //    RD8 : Variant;
   // END_VAR
   // VAR
   //    ident : Byte;
   //    regist : Bool;
   //    flanke : Bool;
   //    progtest : Bool;
   //    err_cls_cod : Word;
   //    err_stat : Word;
   //    s_fifoRef : UInt;
   //    s_Reserved1 : Word;
   //    s_Reserved2 : DWord;
   //    s_Reserved3 : DWord;
   // END_VAR
BEGIN
END_DATA_BLOCK

DATA_BLOCK "LBP_ReadVar_DB_Axis08_W"   // DB4108
// stored: AutoNumber false, InstanceOfName LBP_ReadVar, InstanceOfType FB
"LBP_ReadVar"
   // VAR_INPUT
   //    Req : Bool;
   //    NumVar : Int;
   //    Addr1 : Variant;
   //    Unit1 : Byte;
   //    Column1 : Word;
   //    Line1 : Word;
   //    Addr2 : Variant;
   //    Unit2 : Byte;
   //    Column2 : Word;
   //    Line2 : Word;
   //    Addr3 : Variant;
   //    Unit3 : Byte;
   //    Column3 : Word;
   //    Line3 : Word;
   //    Addr4 : Variant;
   //    Unit4 : Byte;
   //    Column4 : Word;
   //    Line4 : Word;
   //    Addr5 : Variant;
   //    Unit5 : Byte;
   //    Column5 : Word;
   //    Line5 : Word;
   //    Addr6 : Variant;
   //    Unit6 : Byte;
   //    Column6 : Word;
   //    Line6 : Word;
   //    Addr7 : Variant;
   //    Unit7 : Byte;
   //    Column7 : Word;
   //    Line7 : Word;
   //    Addr8 : Variant;
   //    Unit8 : Byte;
   //    Column8 : Word;
   //    Line8 : Word;
   // END_VAR
   // VAR_OUTPUT
   //    Error : Bool;
   //    NDR : Bool;
   //    State : Word;
   // END_VAR
   // VAR_IN_OUT
   //    RD1 : Variant;
   //    RD2 : Variant;
   //    RD3 : Variant;
   //    RD4 : Variant;
   //    RD5 : Variant;
   //    RD6 : Variant;
   //    RD7 : Variant;
   //    RD8 : Variant;
   // END_VAR
   // VAR
   //    ident : Byte;
   //    regist : Bool;
   //    flanke : Bool;
   //    progtest : Bool;
   //    err_cls_cod : Word;
   //    err_stat : Word;
   //    s_fifoRef : UInt;
   //    s_Reserved1 : Word;
   //    s_Reserved2 : DWord;
   //    s_Reserved3 : DWord;
   // END_VAR
BEGIN
END_DATA_BLOCK

DATA_BLOCK "LBP_ReadVar_DB_Axis09_ZL"   // DB4105
// stored: AutoNumber false, InstanceOfName LBP_ReadVar, InstanceOfType FB
"LBP_ReadVar"
   // VAR_INPUT
   //    Req : Bool;
   //    NumVar : Int;
   //    Addr1 : Variant;
   //    Unit1 : Byte;
   //    Column1 : Word;
   //    Line1 : Word;
   //    Addr2 : Variant;
   //    Unit2 : Byte;
   //    Column2 : Word;
   //    Line2 : Word;
   //    Addr3 : Variant;
   //    Unit3 : Byte;
   //    Column3 : Word;
   //    Line3 : Word;
   //    Addr4 : Variant;
   //    Unit4 : Byte;
   //    Column4 : Word;
   //    Line4 : Word;
   //    Addr5 : Variant;
   //    Unit5 : Byte;
   //    Column5 : Word;
   //    Line5 : Word;
   //    Addr6 : Variant;
   //    Unit6 : Byte;
   //    Column6 : Word;
   //    Line6 : Word;
   //    Addr7 : Variant;
   //    Unit7 : Byte;
   //    Column7 : Word;
   //    Line7 : Word;
   //    Addr8 : Variant;
   //    Unit8 : Byte;
   //    Column8 : Word;
   //    Line8 : Word;
   // END_VAR
   // VAR_OUTPUT
   //    Error : Bool;
   //    NDR : Bool;
   //    State : Word;
   // END_VAR
   // VAR_IN_OUT
   //    RD1 : Variant;
   //    RD2 : Variant;
   //    RD3 : Variant;
   //    RD4 : Variant;
   //    RD5 : Variant;
   //    RD6 : Variant;
   //    RD7 : Variant;
   //    RD8 : Variant;
   // END_VAR
   // VAR
   //    ident : Byte;
   //    regist : Bool;
   //    flanke : Bool;
   //    progtest : Bool;
   //    err_cls_cod : Word;
   //    err_stat : Word;
   //    s_fifoRef : UInt;
   //    s_Reserved1 : Word;
   //    s_Reserved2 : DWord;
   //    s_Reserved3 : DWord;
   // END_VAR
BEGIN
END_DATA_BLOCK

DATA_BLOCK "DB_ChillerSMC"   // DB541
// stored: AutoNumber false, InstanceOfName FB_ChillerSMC, InstanceOfType FB
"FB_ChillerSMC"
BEGIN
END_DATA_BLOCK

DATA_BLOCK "DB_ChillerTermotek"   // DB540
// stored: AutoNumber false, InstanceOfName FB_ChillerTermotek, InstanceOfType FB
"FB_ChillerTermotek"
BEGIN
END_DATA_BLOCK

DATA_BLOCK "CONT_C_Clim_DB"   // DB2251
// stored: InstanceOfName CONT_C, OfSystemLibElement CONT_C, OfSystemLibVersion 1.1
CONT_C   // technology object, version 1.1
   // VAR_INPUT
   //    COM_RST : Bool;
   //    MAN_ON : Bool;
   //    PVPER_ON : Bool;
   //    P_SEL : Bool;
   //    I_SEL : Bool;
   //    INT_HOLD : Bool;
   //    I_ITL_ON : Bool;
   //    D_SEL : Bool;
   //    CYCLE : Time;
   //    SP_INT : Real;
   //    PV_IN : Real;
   //    PV_PER : Word;
   //    MAN : Real;
   //    GAIN : Real;
   //    TI : Time;
   //    TD : Time;
   //    TM_LAG : Time;
   //    DEADB_W : Real;
   //    LMN_HLM : Real;
   //    LMN_LLM : Real;
   //    PV_FAC : Real;
   //    PV_OFF : Real;
   //    LMN_FAC : Real;
   //    LMN_OFF : Real;
   //    I_ITLVAL : Real;
   //    DISV : Real;
   // END_VAR
   // VAR_OUTPUT
   //    LMN : Real;
   //    LMN_PER : Word;
   //    QLMN_HLM : Bool;
   //    QLMN_LLM : Bool;
   //    LMN_P : Real;
   //    LMN_I : Real;
   //    LMN_D : Real;
   //    PV : Real;
   //    ER : Real;
   // END_VAR
   // VAR RETAIN
   //    sInvAlt : Real;
   //    sIanteilAlt : Real;
   //    sRestInt : Real;
   //    sRestDif : Real;
   //    sRueck : Real;
   //    sLmn : Real;
   //    sbArwHLmOn : Bool;
   //    sbArwLLmOn : Bool;
   //    sbILimOn : Bool;
   // END_VAR
BEGIN
END_DATA_BLOCK
